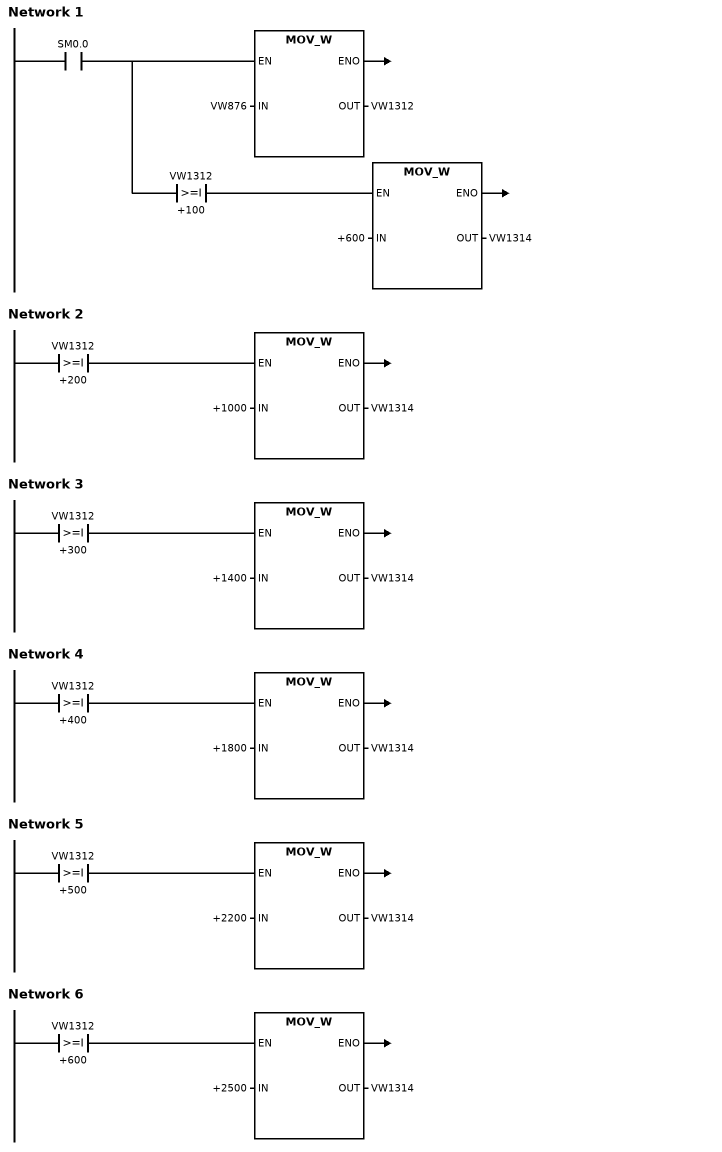
[picture p96: SBR24 networks 1-6]
Network 1
LD     SM0.0
MOVW   VW876, VW1312
AW>=   VW1312, +100
MOVW   +600, VW1314
Network 2
LDW>=  VW1312, +200
MOVW   +1000, VW1314
Network 3
LDW>=  VW1312, +300
MOVW   +1400, VW1314
Network 4
LDW>=  VW1312, +400
MOVW   +1800, VW1314
Network 5
LDW>=  VW1312, +500
MOVW   +2200, VW1314
Network 6
LDW>=  VW1312, +600
MOVW   +2500, VW1314
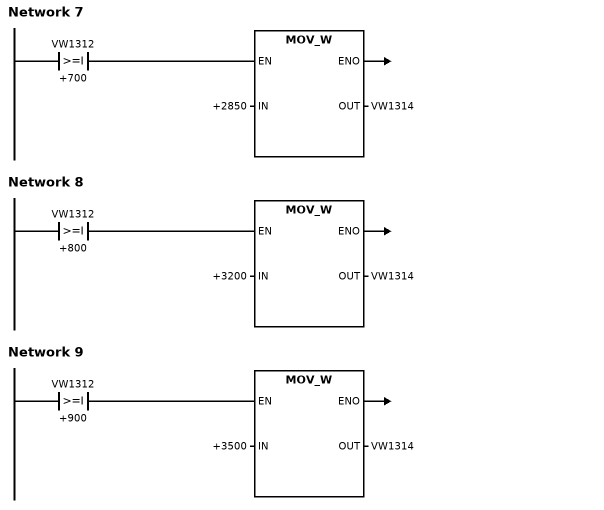
Network 7
LDW>=  VW1312, +700
MOVW   +2850, VW1314
Network 8
LDW>=  VW1312, +800
MOVW   +3200, VW1314
Network 9
LDW>=  VW1312, +900
MOVW   +3500, VW1314
END_SUBROUTINE_BLOCK

SUBROUTINE_BLOCK SprayMotorSpeedChange:SBR25
TITLE=
BEGIN
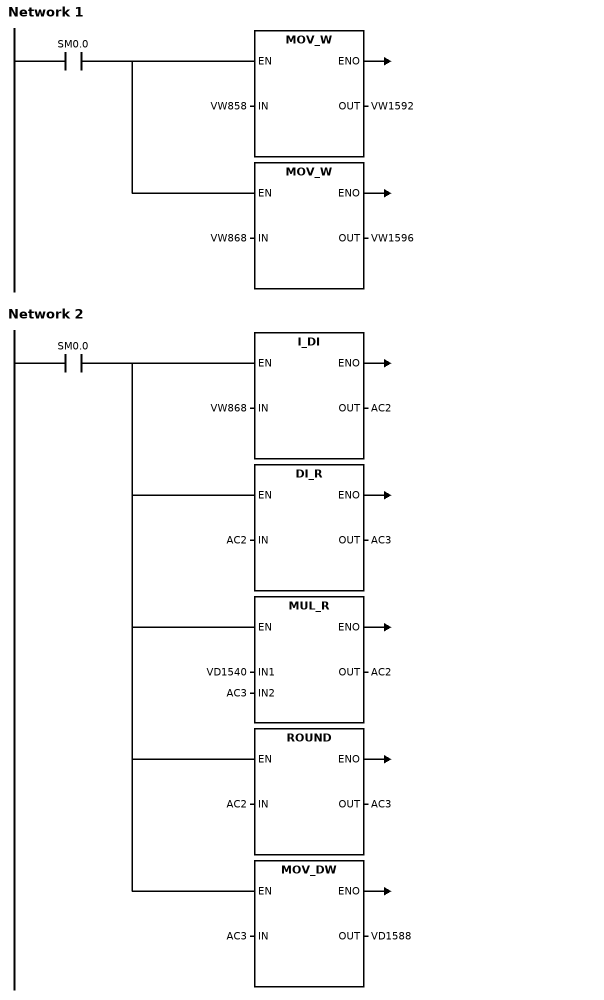
Network 1
LD     SM0.0
MOVW   VW858, VW1592
MOVW   VW868, VW1596
Network 2
LD     SM0.0
ITD    VW868, AC2
DTR    AC2, AC3
MOVR   VD1540, AC2
*R     AC3, AC2
ROUND  AC2, AC3
MOVD   AC3, VD1588
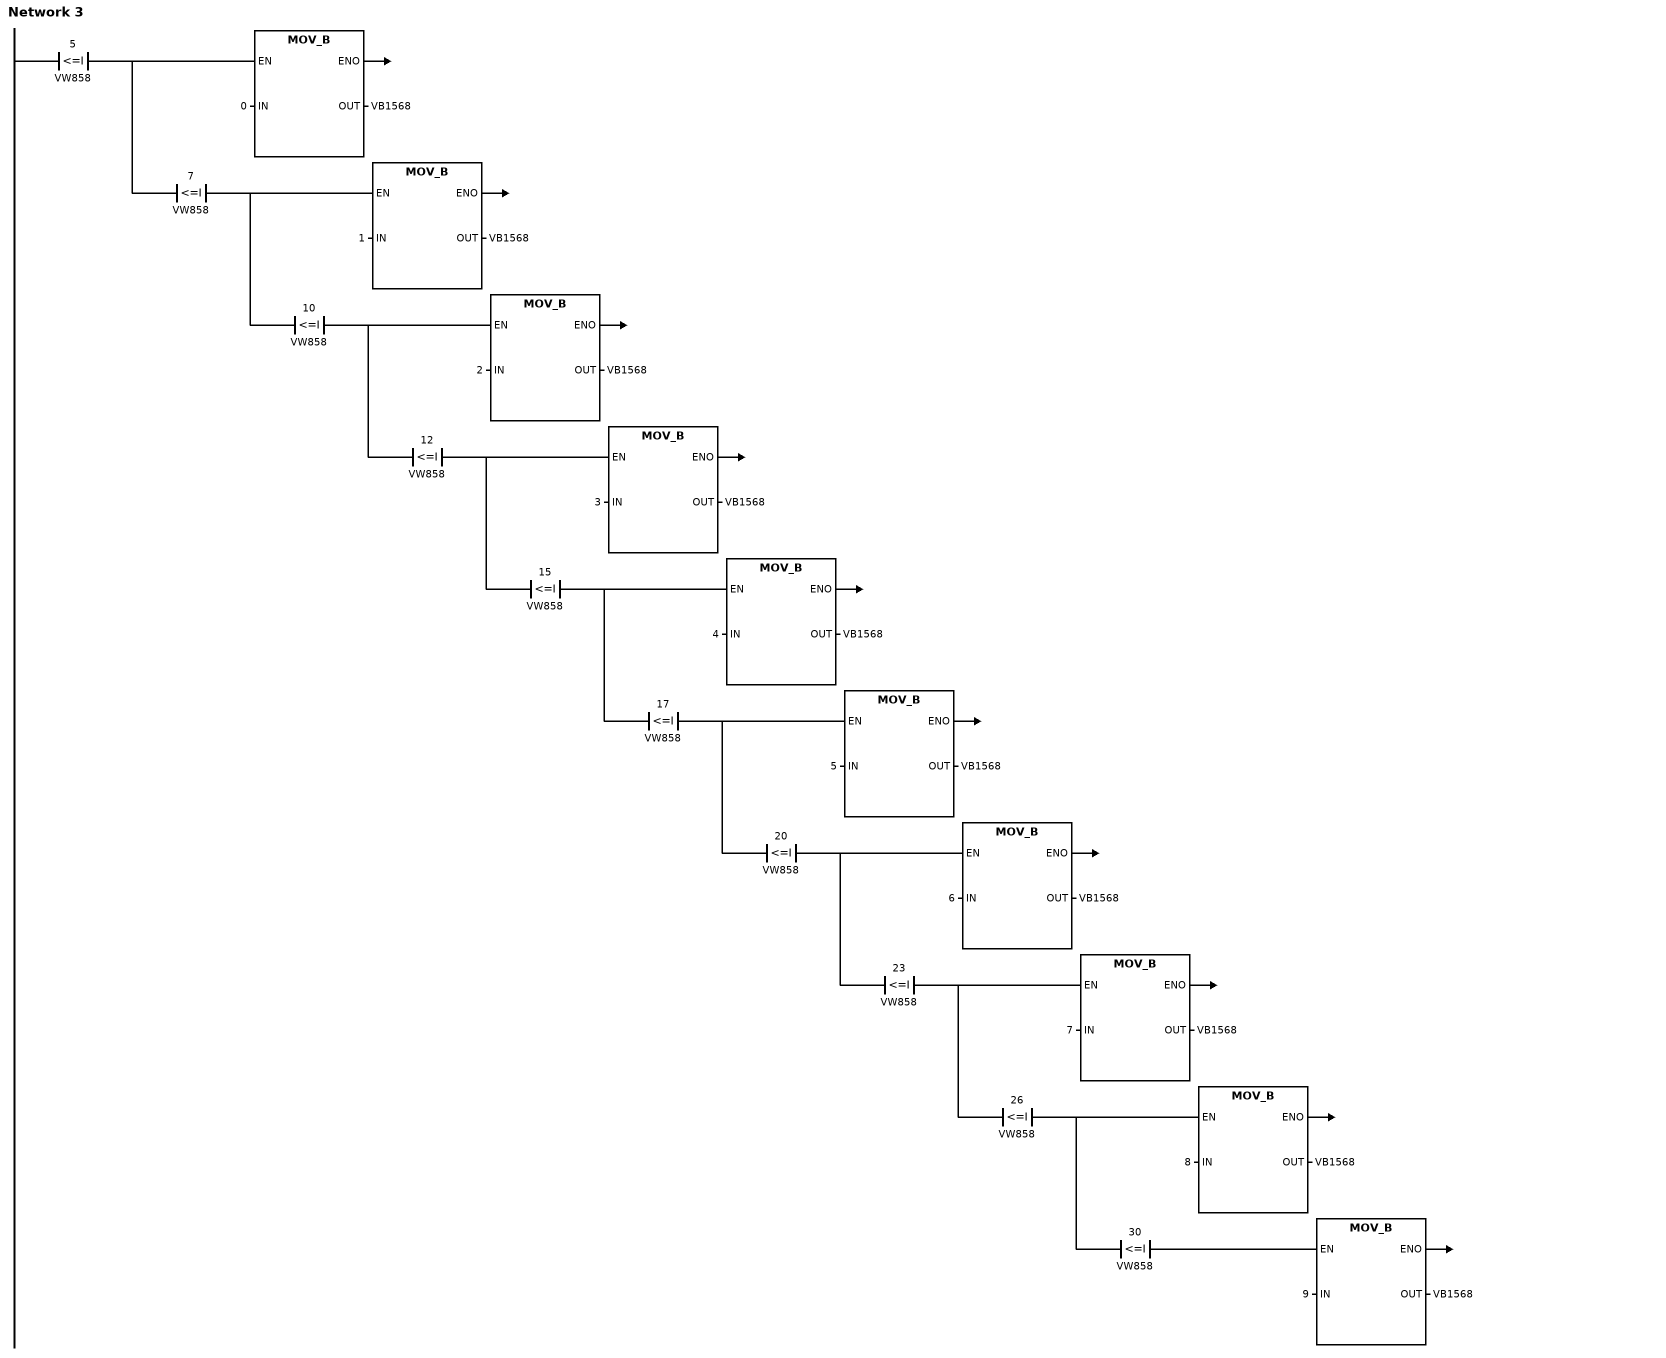
Network 3
LDW<=  5, VW858
MOVB   0, VB1568
AW<=   7, VW858
MOVB   1, VB1568
AW<=   10, VW858
MOVB   2, VB1568
AW<=   12, VW858
MOVB   3, VB1568
AW<=   15, VW858
MOVB   4, VB1568
AW<=   17, VW858
MOVB   5, VB1568
AW<=   20, VW858
MOVB   6, VB1568
AW<=   23, VW858
MOVB   7, VB1568
AW<=   26, VW858
MOVB   8, VB1568
AW<=   30, VW858
MOVB   9, VB1568
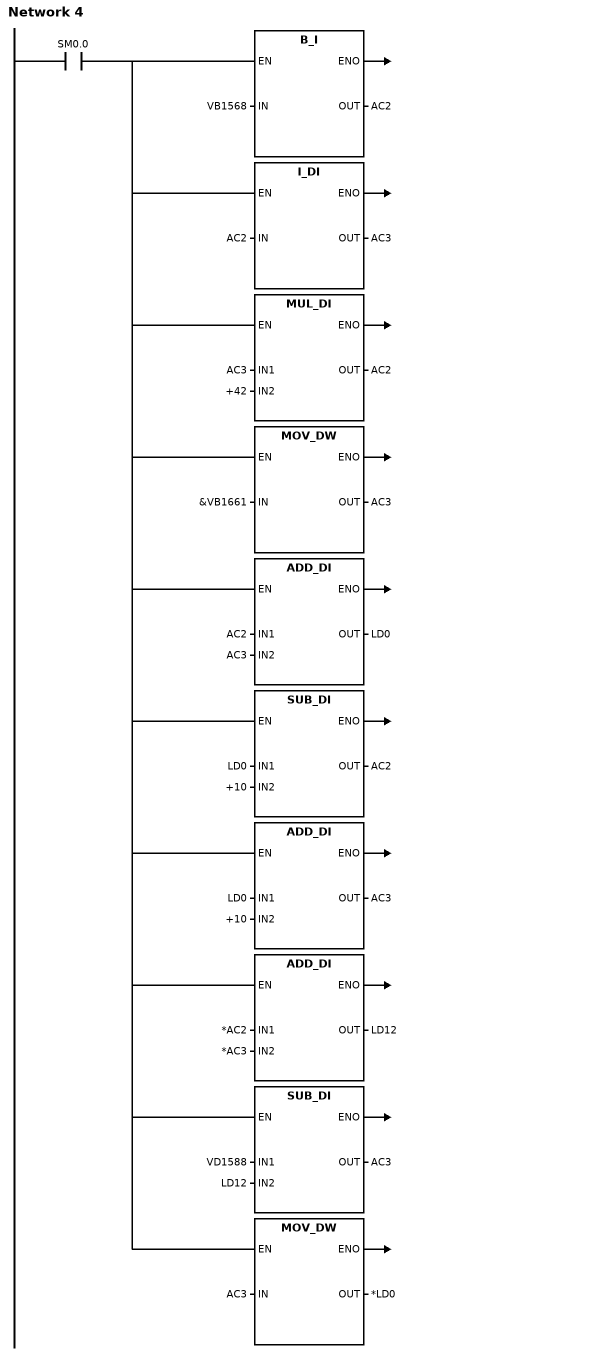
Network 4
LD     SM0.0
BTI    VB1568, AC2
ITD    AC2, AC3
MOVD   AC3, AC2
*D     +42, AC2
MOVD   &VB1661, AC3
MOVD   AC2, LD0
+D     AC3, LD0
MOVD   LD0, AC2
-D     +10, AC2
MOVD   LD0, AC3
+D     +10, AC3
MOVD   *AC2, LD12
+D     *AC3, LD12
MOVD   VD1588, AC3
-D     LD12, AC3
MOVD   AC3, *LD0
END_SUBROUTINE_BLOCK

// SBR26: protected block, not included

// SBR27: protected block, not included

// SBR28: protected block, not included

SUBROUTINE_BLOCK SysConfigure:SBR29
TITLE=SUBROUTINE COMMENTS
BEGIN
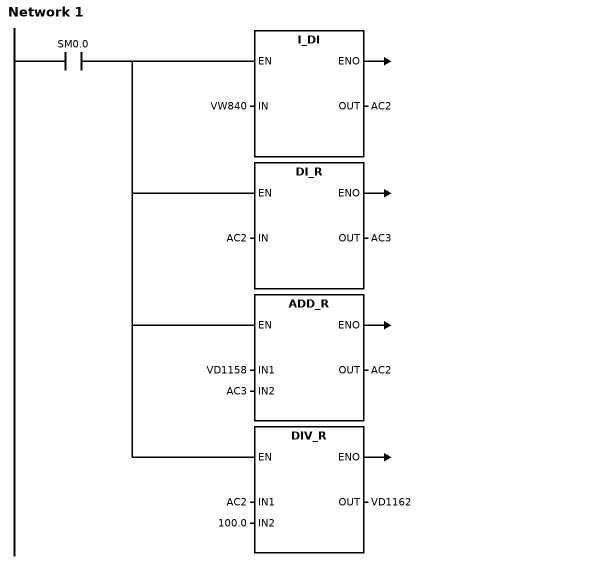
Network 1
LD     SM0.0
ITD    VW840, AC2
DTR    AC2, AC3
MOVR   VD1158, AC2
+R     AC3, AC2
MOVR   AC2, VD1162
/R     100.0, VD1162
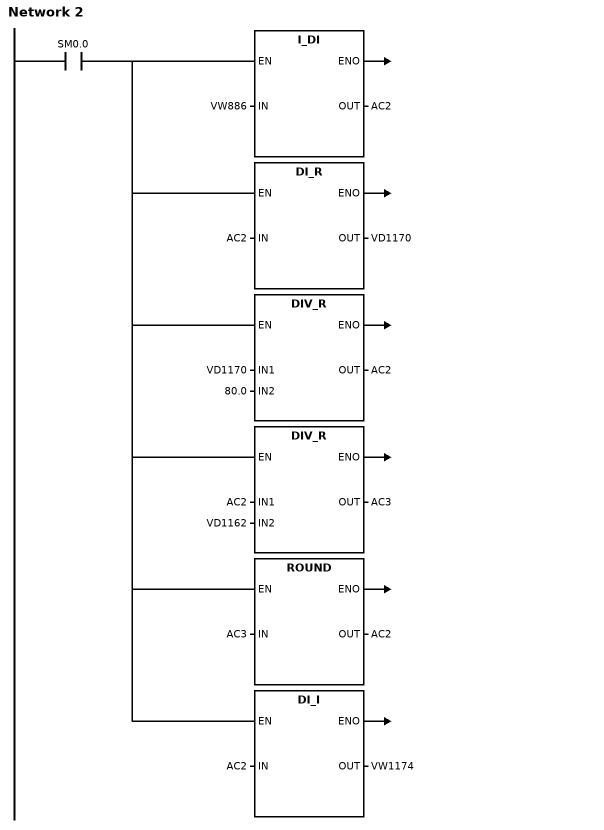
Network 2
LD     SM0.0
ITD    VW886, AC2
DTR    AC2, VD1170
MOVR   VD1170, AC2
/R     80.0, AC2
MOVR   AC2, AC3
/R     VD1162, AC3
ROUND  AC3, AC2
DTI    AC2, VW1174
END_SUBROUTINE_BLOCK

SUBROUTINE_BLOCK MyPID_M1:SBR30
TITLE=SUBROUTINE COMMENTS
VAR_INPUT
iSV:INT;	// LW0 
iPV:INT;	// LW2 
iKT:INT;	// LW4 
iKP:INT;	// LW6 
iKI:INT;	// LW8 
iKD:INT;	// LW10 
iOffset:INT;	// LW12 
pDataSave:DWORD;	// LD14 
END_VAR
VAR_OUTPUT
iPWM_1:INT;	// LW18 
chTrend:BYTE;	// LB20 
END_VAR
BEGIN
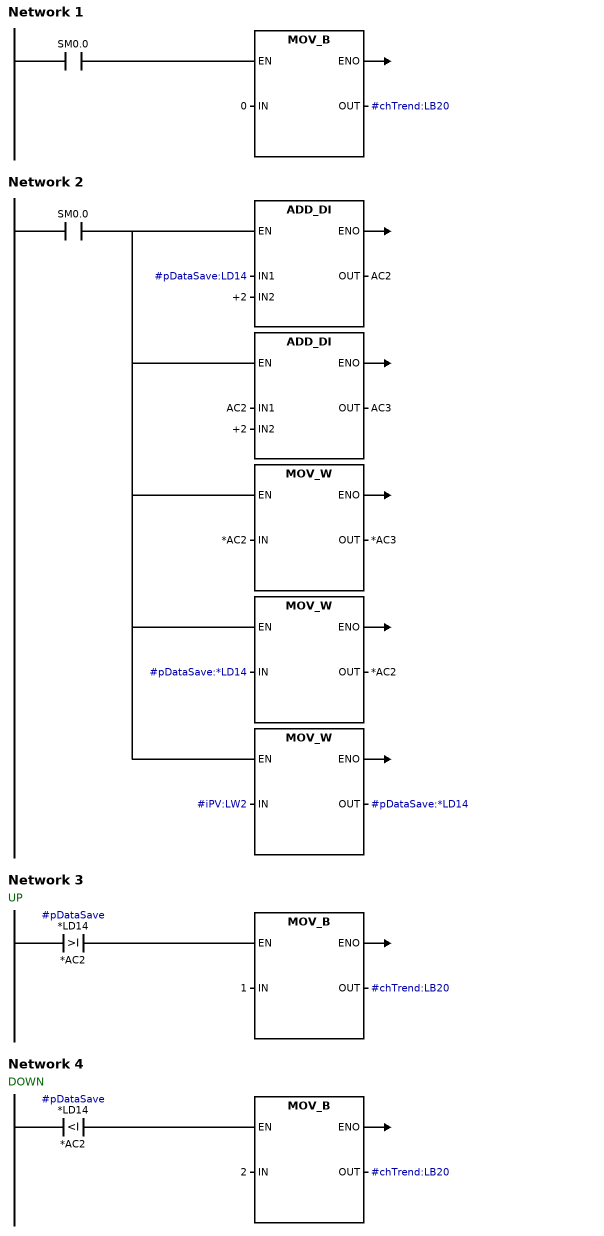
Network 1
LD     SM0.0
MOVB   0, #chTrend:LB20
Network 2
LD     SM0.0
MOVD   #pDataSave:LD14, AC2
+D     +2, AC2
MOVD   AC2, AC3
+D     +2, AC3
MOVW   *AC2, *AC3
MOVW   *#pDataSave:LD14, *AC2
MOVW   #iPV:LW2, *#pDataSave:LD14
Network 3
// UP
LDW>   *#pDataSave:LD14, *AC2
MOVB   1, #chTrend:LB20
Network 4
// DOWN
LDW<   *#pDataSave:LD14, *AC2
MOVB   2, #chTrend:LB20
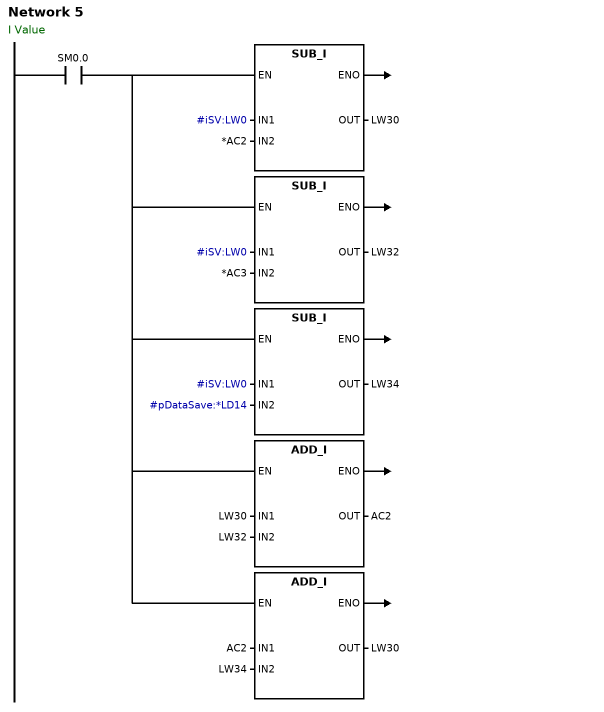
Network 5
// I Value
LD     SM0.0
MOVW   #iSV:LW0, LW30
-I     *AC2, LW30
MOVW   #iSV:LW0, LW32
-I     *AC3, LW32
MOVW   #iSV:LW0, LW34
-I     *#pDataSave:LD14, LW34
MOVW   LW30, AC2
+I     LW32, AC2
MOVW   AC2, LW30
+I     LW34, LW30
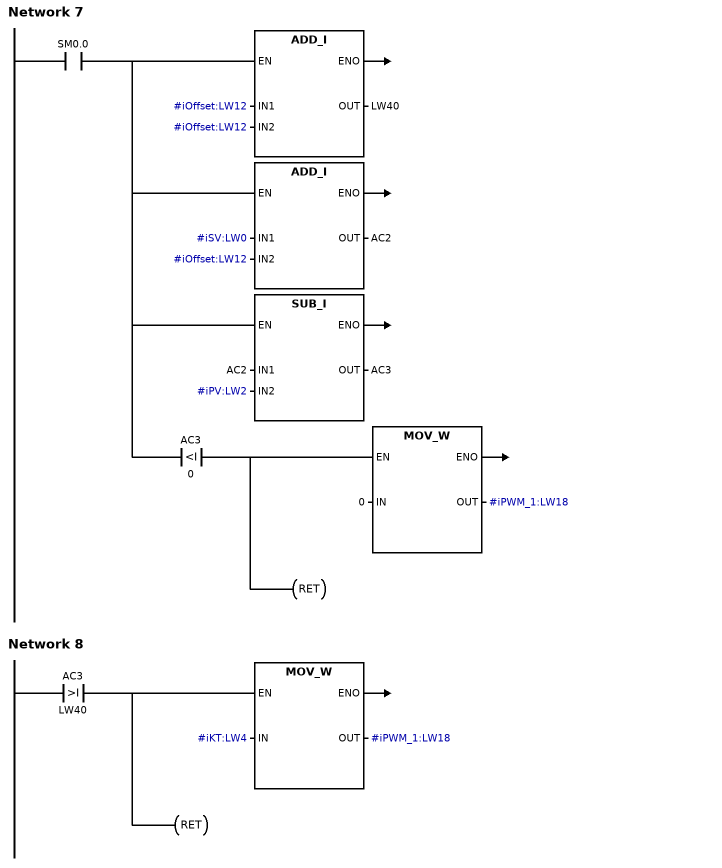
Network 7
LD     SM0.0
MOVW   #iOffset:LW12, LW40
+I     #iOffset:LW12, LW40
MOVW   #iSV:LW0, AC2
+I     #iOffset:LW12, AC2
MOVW   AC2, AC3
-I     #iPV:LW2, AC3
AW<    AC3, 0
MOVW   0, #iPWM_1:LW18
CRET
Network 8
LDW>   AC3, LW40
MOVW   #iKT:LW4, #iPWM_1:LW18
CRET
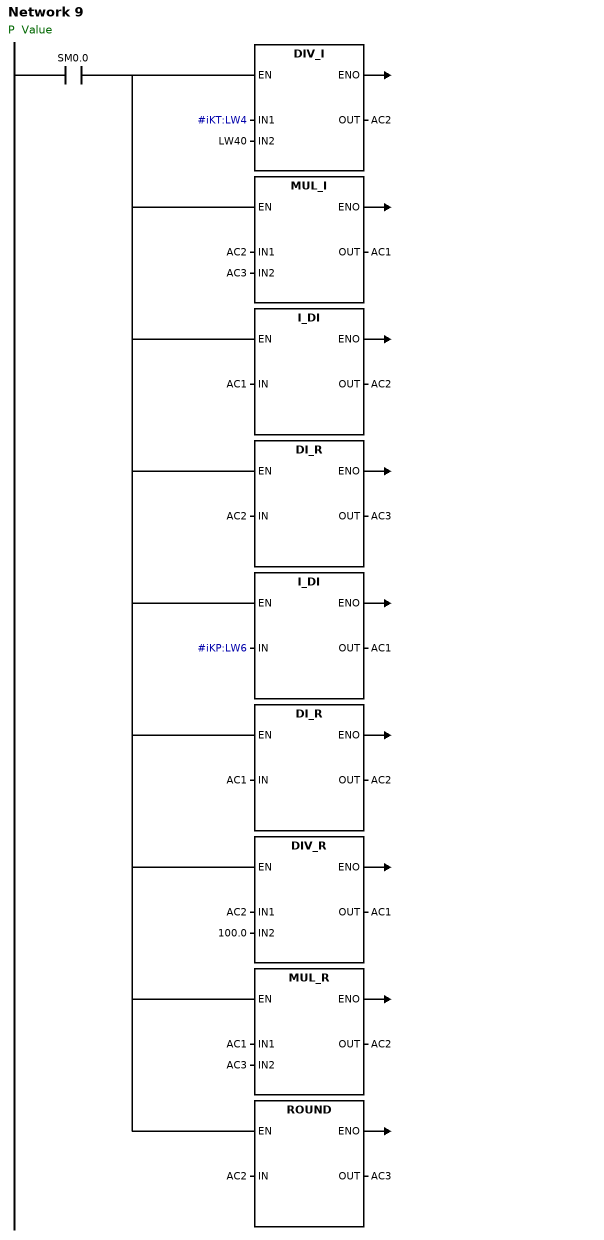
Network 9
// P  Value
LD     SM0.0
MOVW   #iKT:LW4, AC2
/I     LW40, AC2
MOVW   AC2, AC1
*I     AC3, AC1
ITD    AC1, AC2
DTR    AC2, AC3
ITD    #iKP:LW6, AC1
DTR    AC1, AC2
MOVR   AC2, AC1
/R     100.0, AC1
MOVR   AC1, AC2
*R     AC3, AC2
ROUND  AC2, AC3
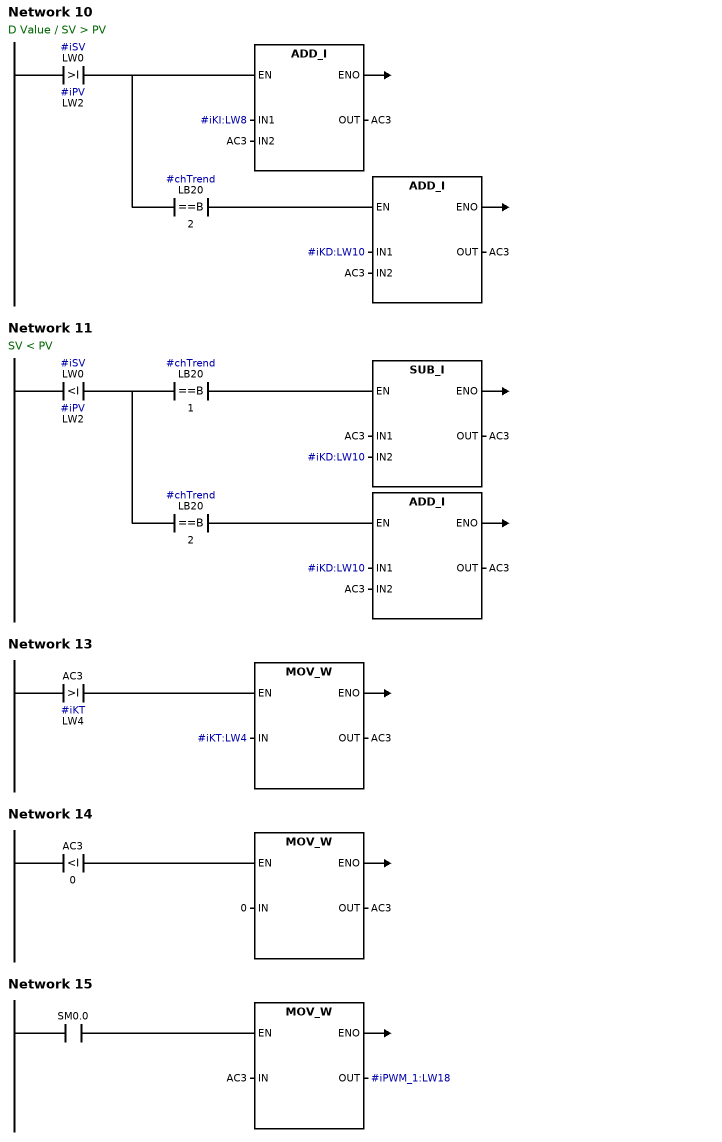
Network 10
// D Value
// SV > PV
LDW>   #iSV:LW0, #iPV:LW2
+I     #iKI:LW8, AC3
AB=    #chTrend:LB20, 2
+I     #iKD:LW10, AC3
Network 11
// SV < PV
LDW<   #iSV:LW0, #iPV:LW2
LPS
AB=    #chTrend:LB20, 1
-I     #iKD:LW10, AC3
LPP
AB=    #chTrend:LB20, 2
+I     #iKD:LW10, AC3
Network 12
// I????
Network 13
LDW>   AC3, #iKT:LW4
MOVW   #iKT:LW4, AC3
Network 14
LDW<   AC3, 0
MOVW   0, AC3
Network 15
LD     SM0.0
MOVW   AC3, #iPWM_1:LW18
END_SUBROUTINE_BLOCK

SUBROUTINE_BLOCK StopQ1Pulse:SBR31
TITLE=SUBROUTINE COMMENTS
BEGIN
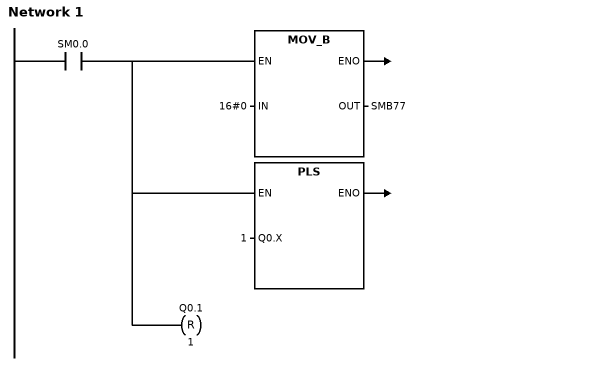
Network 1
LD     SM0.0
MOVB   16#0, SMB77
PLS    1
R      Q0.1, 1
END_SUBROUTINE_BLOCK

SUBROUTINE_BLOCK WidthPulseVB4000_4099:SBR32
TITLE=SUBROUTINE COMMENTS
VAR_INPUT
iPCBWidth:INT;	// LW0 
iSpeedHz:INT;	// LW2 
END_VAR
BEGIN
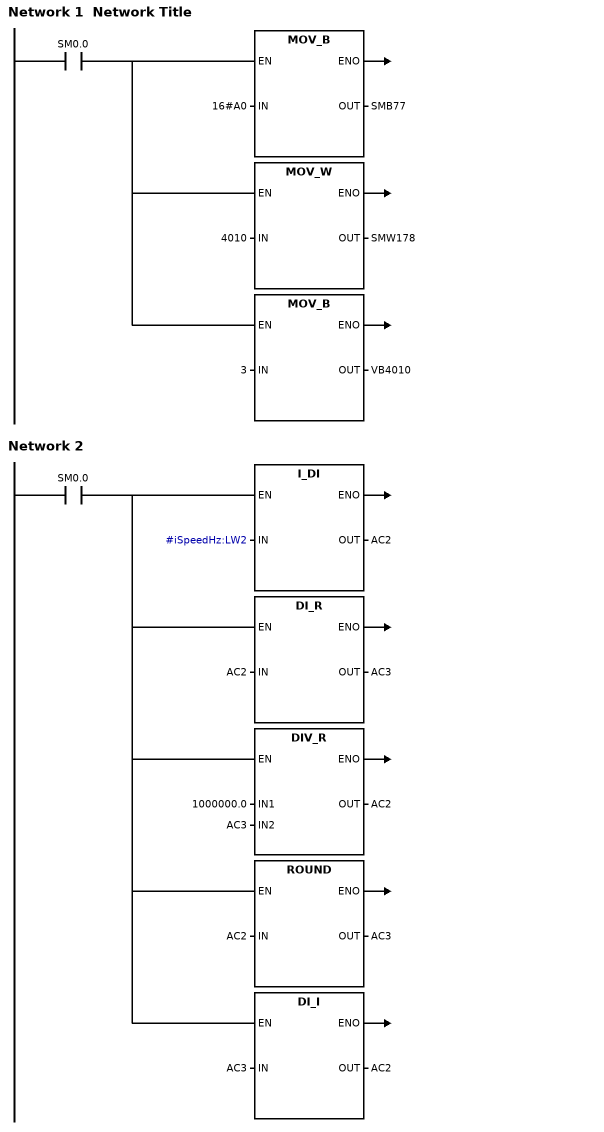
Network 1 // Network Title
LD     SM0.0
MOVB   16#A0, SMB77
MOVW   4010, SMW178
MOVB   3, VB4010
Network 2
LD     SM0.0
ITD    #iSpeedHz:LW2, AC2
DTR    AC2, AC3
MOVR   1000000.0, AC2
/R     AC3, AC2
ROUND  AC2, AC3
DTI    AC3, AC2
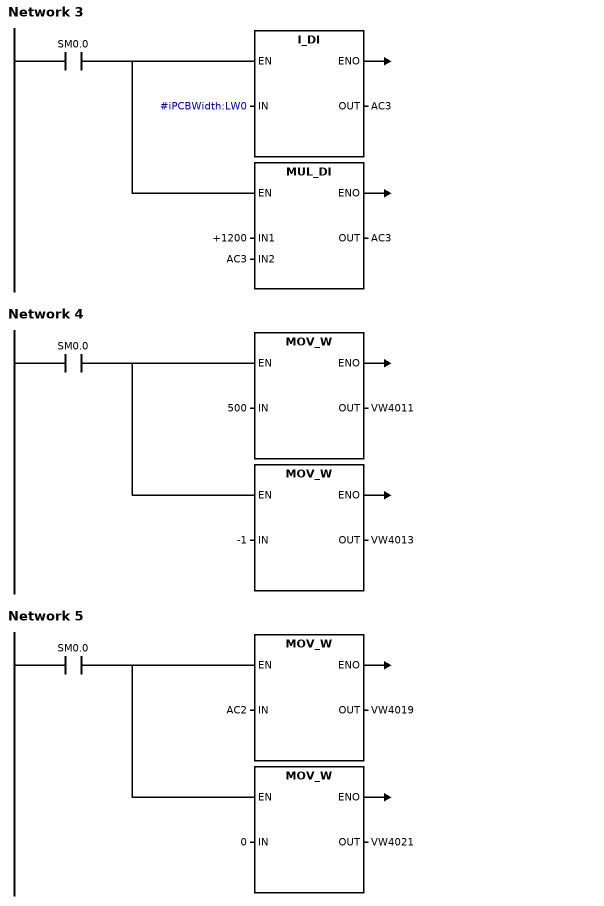
Network 3
LD     SM0.0
ITD    #iPCBWidth:LW0, AC3
*D     +1200, AC3
Network 4
LD     SM0.0
MOVW   500, VW4011
MOVW   -1, VW4013
Network 5
LD     SM0.0
MOVW   AC2, VW4019
MOVW   0, VW4021
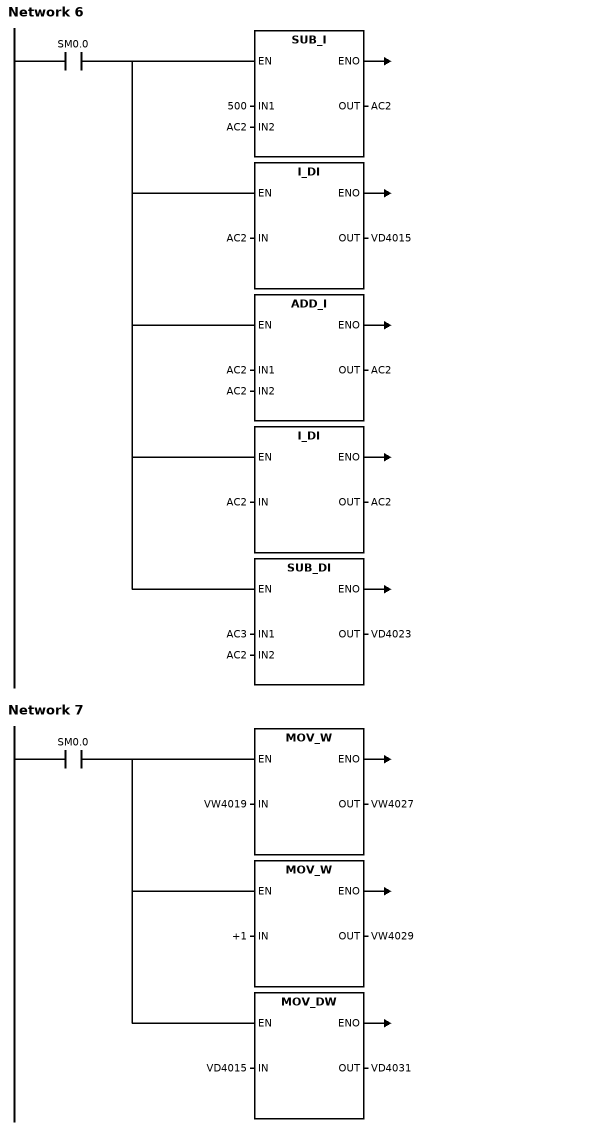
Network 6
LD     SM0.0
INVW   AC2
INCW   AC2
+I     500, AC2
ITD    AC2, VD4015
+I     AC2, AC2
ITD    AC2, AC2
MOVD   AC3, VD4023
-D     AC2, VD4023
Network 7
LD     SM0.0
MOVW   VW4019, VW4027
MOVW   +1, VW4029
MOVD   VD4015, VD4031
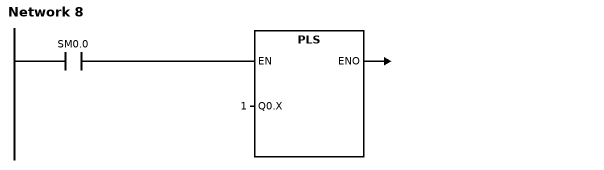
Network 8
LD     SM0.0
PLS    1
END_SUBROUTINE_BLOCK

SUBROUTINE_BLOCK TimerFlagVB600_699:SBR33
TITLE=SUBROUTINE COMMENTS
BEGIN
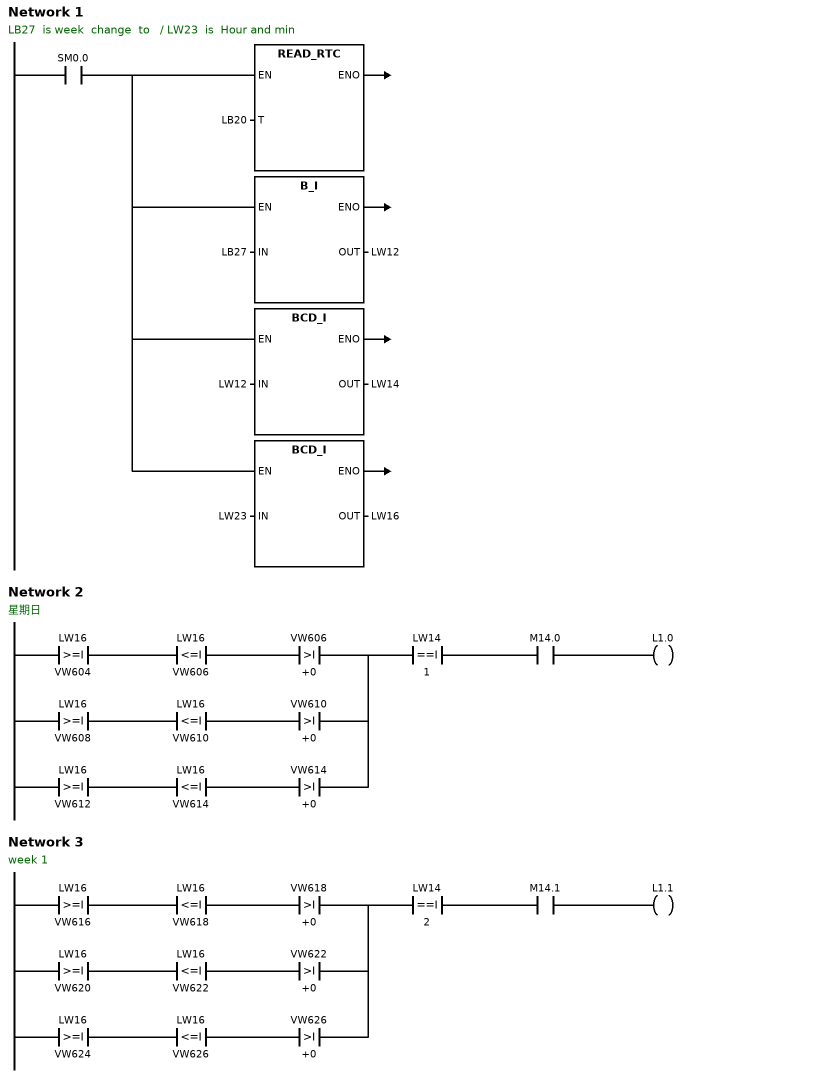
Network 1
// LB27  is week  change  to  
// LW23  is  Hour and min
LD     SM0.0
TODR   LB20
BTI    LB27, LW12
MOVW   LW12, LW14
BCDI   LW14
MOVW   LW23, LW16
BCDI   LW16
Network 2
// 星期日
LDW>=  LW16, VW604
AW<=   LW16, VW606
AW>    VW606, +0
LDW>=  LW16, VW608
AW<=   LW16, VW610
AW>    VW610, +0
OLD
LDW>=  LW16, VW612
AW<=   LW16, VW614
AW>    VW614, +0
OLD
AW=    LW14, 1
A      M14.0
=      L1.0
Network 3
// week 1
LDW>=  LW16, VW616
AW<=   LW16, VW618
AW>    VW618, +0
LDW>=  LW16, VW620
AW<=   LW16, VW622
AW>    VW622, +0
OLD
LDW>=  LW16, VW624
AW<=   LW16, VW626
AW>    VW626, +0
OLD
AW=    LW14, 2
A      M14.1
=      L1.1
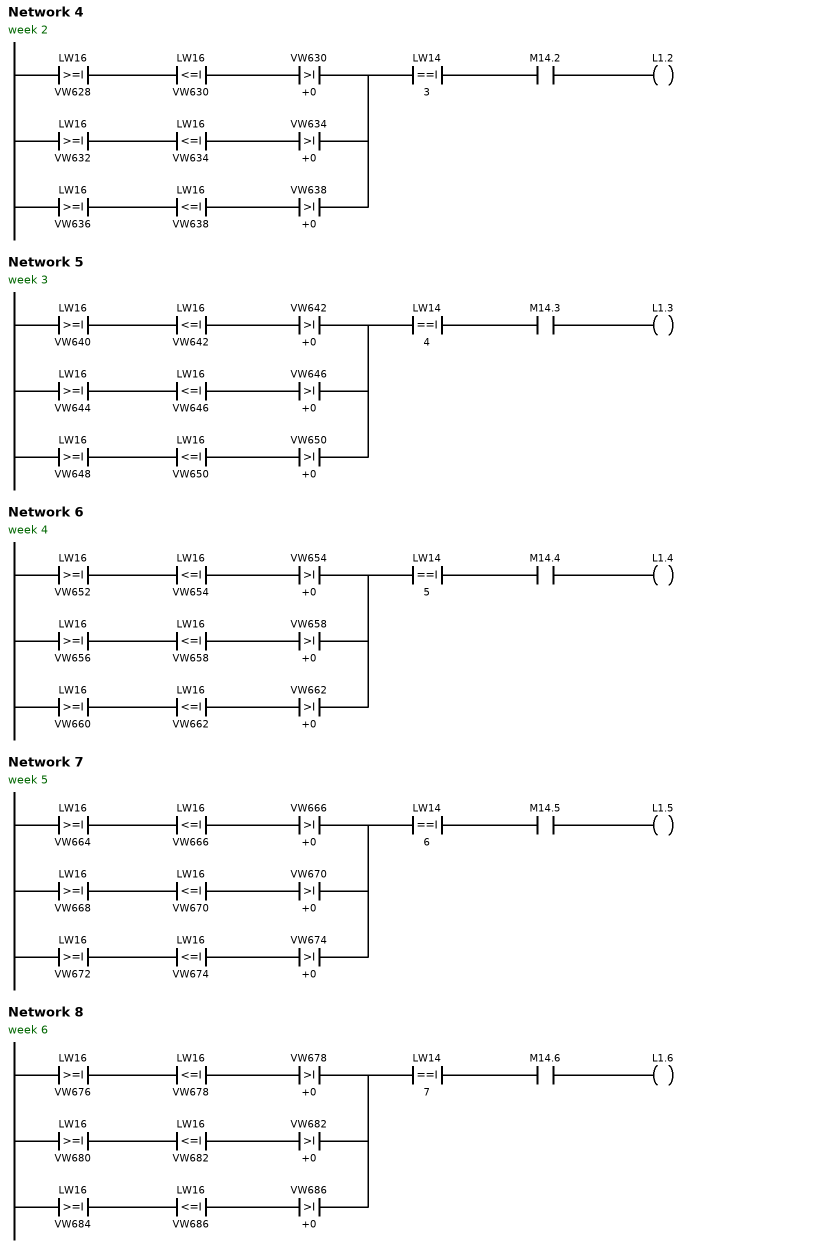
Network 4
// week 2
LDW>=  LW16, VW628
AW<=   LW16, VW630
AW>    VW630, +0
LDW>=  LW16, VW632
AW<=   LW16, VW634
AW>    VW634, +0
OLD
LDW>=  LW16, VW636
AW<=   LW16, VW638
AW>    VW638, +0
OLD
AW=    LW14, 3
A      M14.2
=      L1.2
Network 5
// week 3
LDW>=  LW16, VW640
AW<=   LW16, VW642
AW>    VW642, +0
LDW>=  LW16, VW644
AW<=   LW16, VW646
AW>    VW646, +0
OLD
LDW>=  LW16, VW648
AW<=   LW16, VW650
AW>    VW650, +0
OLD
AW=    LW14, 4
A      M14.3
=      L1.3
Network 6
// week 4
LDW>=  LW16, VW652
AW<=   LW16, VW654
AW>    VW654, +0
LDW>=  LW16, VW656
AW<=   LW16, VW658
AW>    VW658, +0
OLD
LDW>=  LW16, VW660
AW<=   LW16, VW662
AW>    VW662, +0
OLD
AW=    LW14, 5
A      M14.4
=      L1.4
Network 7
// week 5
LDW>=  LW16, VW664
AW<=   LW16, VW666
AW>    VW666, +0
LDW>=  LW16, VW668
AW<=   LW16, VW670
AW>    VW670, +0
OLD
LDW>=  LW16, VW672
AW<=   LW16, VW674
AW>    VW674, +0
OLD
AW=    LW14, 6
A      M14.5
=      L1.5
Network 8
// week 6
LDW>=  LW16, VW676
AW<=   LW16, VW678
AW>    VW678, +0
LDW>=  LW16, VW680
AW<=   LW16, VW682
AW>    VW682, +0
OLD
LDW>=  LW16, VW684
AW<=   LW16, VW686
AW>    VW686, +0
OLD
AW=    LW14, 7
A      M14.6
=      L1.6
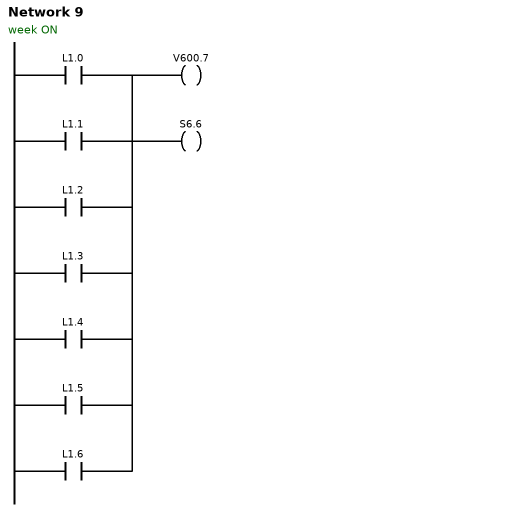
Network 9
// week ON
LD     L1.0
O      L1.1
O      L1.2
O      L1.3
O      L1.4
O      L1.5
O      L1.6
=      V600.7
=      S6.6
END_SUBROUTINE_BLOCK

SUBROUTINE_BLOCK Preheart_equalize:SBR34
TITLE=WaveSpewWagVB1300_1319//T160_T164
BEGIN
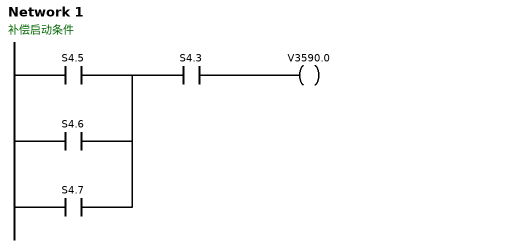
Network 1
// 补偿启动条件
LD     S4.5
O      S4.6
O      S4.7
A      S4.3
=      V3590.0
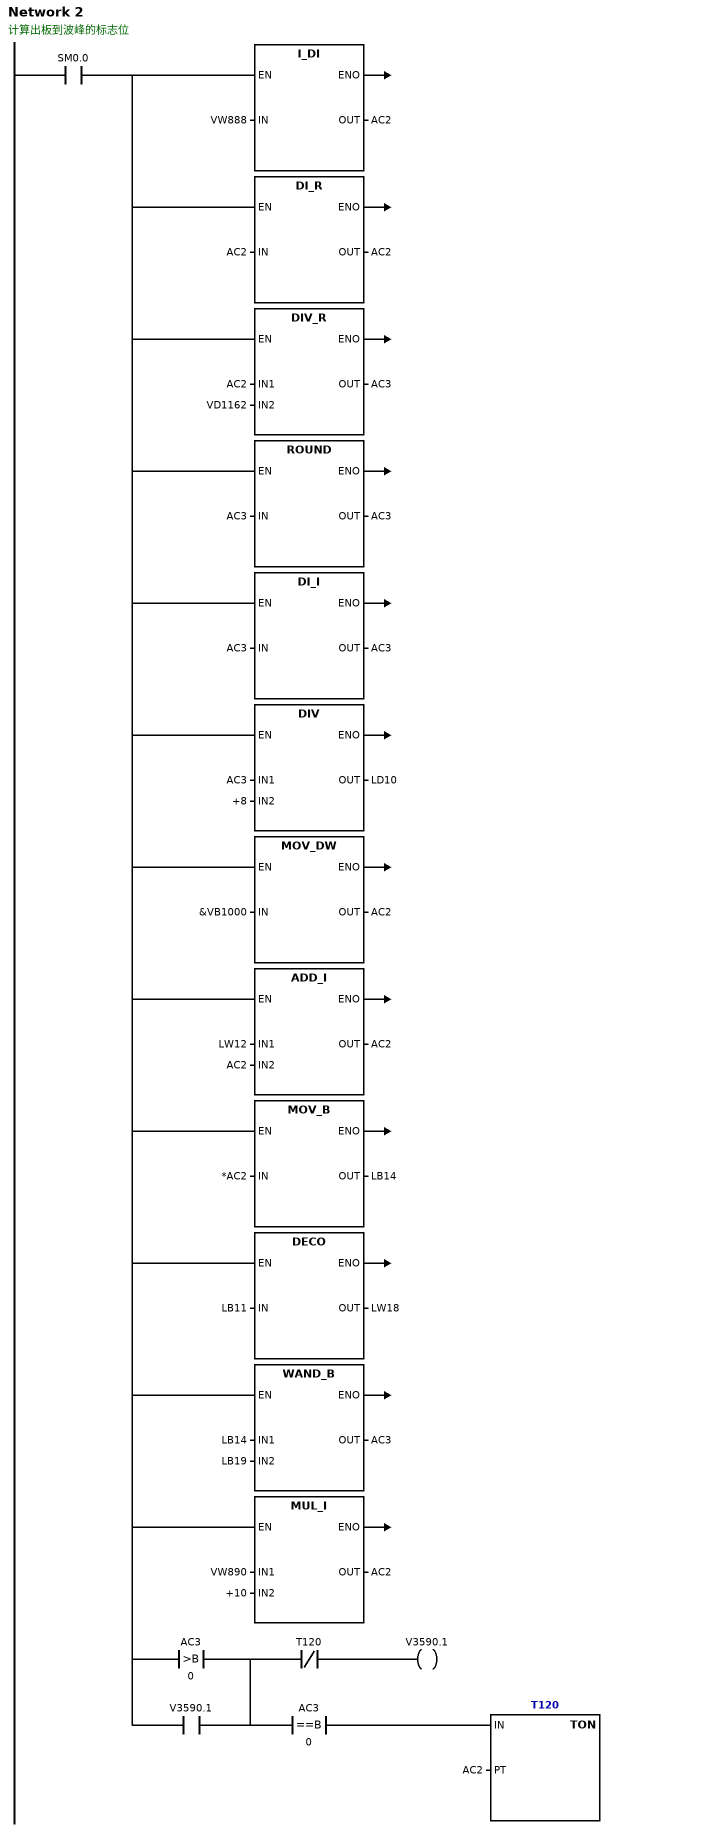
Network 2
// 计算出板到波峰的标志位
LD     SM0.0
ITD    VW888, AC2
DTR    AC2, AC2
MOVR   AC2, AC3
/R     VD1162, AC3
ROUND  AC3, AC3
DTI    AC3, AC3
MOVW   AC3, LW12
DIV    +8, LD10
MOVD   &VB1000, AC2
+I     LW12, AC2
MOVB   *AC2, LB14
DECO   LB11, LW18
MOVB   LB14, AC3
ANDB   LB19, AC3
MOVW   VW890, AC2
*I     +10, AC2
LDB>   AC3, 0
O      V3590.1
ALD
LPS
AN     T120
=      V3590.1
LPP
AB=    AC3, 0
TON    T120, AC2
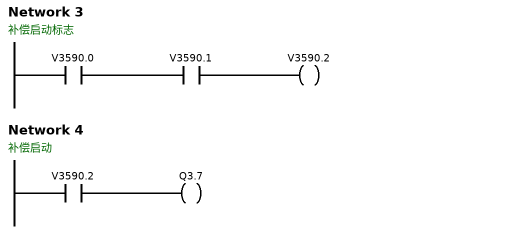
Network 3
// 补偿启动标志
LD     V3590.0
A      V3590.1
=      V3590.2
Network 4
// 补偿启动
LD     V3590.2
=      Q3.7
Network 5 // 网络标题
// 网络注释
Network 15 // 网络标题
// 网络注释
Network 25 // Network Title
// Network Comment
END_SUBROUTINE_BLOCK

SUBROUTINE_BLOCK PCB_Block:SBR45
TITLE=子程序注释
BEGIN
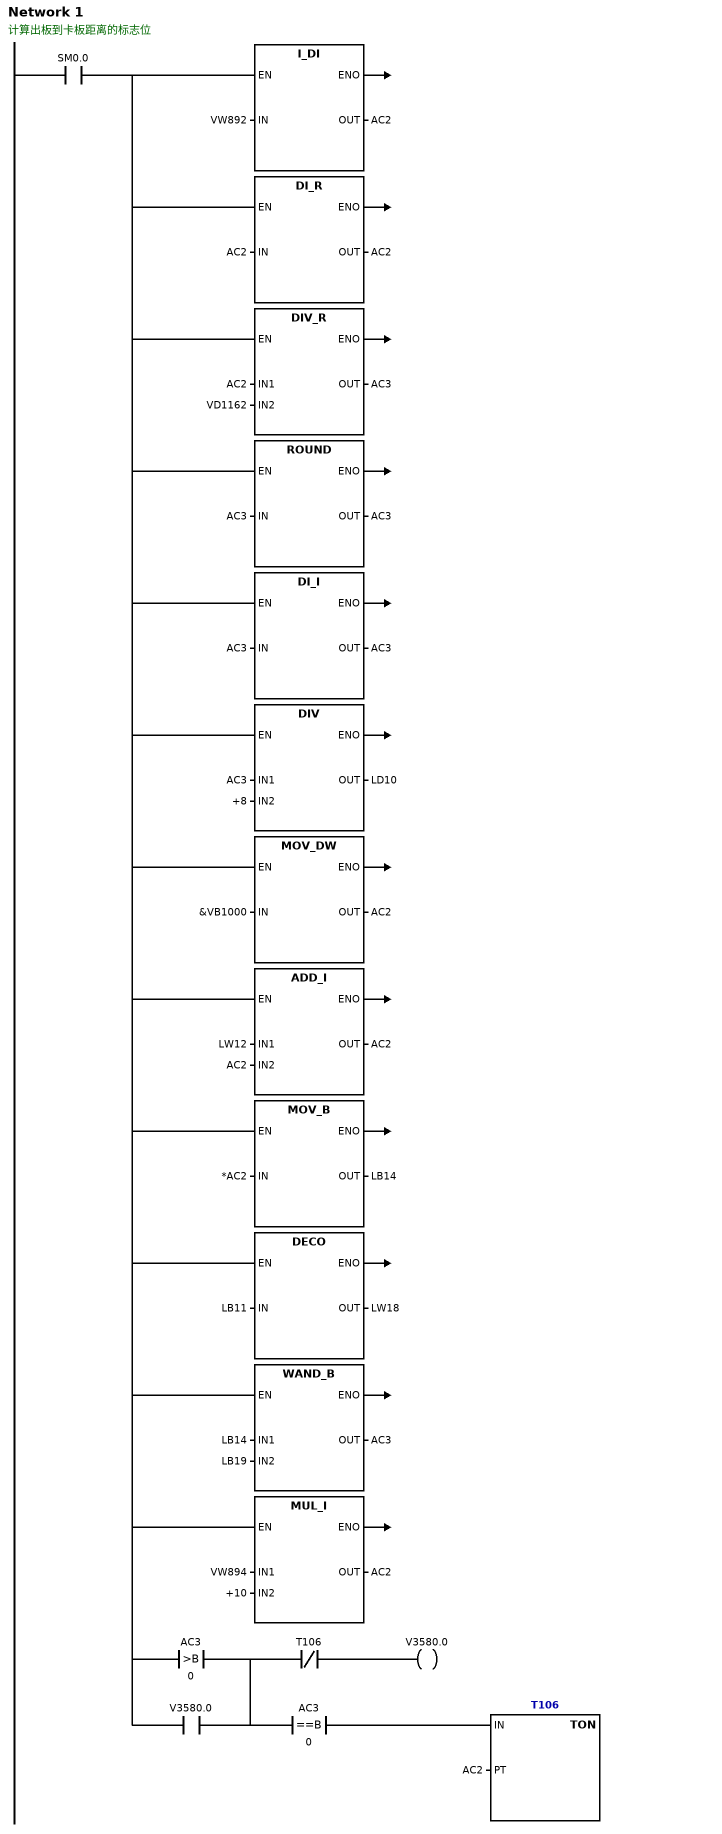
Network 1
// 计算出板到卡板距离的标志位
LD     SM0.0
ITD    VW892, AC2
DTR    AC2, AC2
MOVR   AC2, AC3
/R     VD1162, AC3
ROUND  AC3, AC3
DTI    AC3, AC3
MOVW   AC3, LW12
DIV    +8, LD10
MOVD   &VB1000, AC2
+I     LW12, AC2
MOVB   *AC2, LB14
DECO   LB11, LW18
MOVB   LB14, AC3
ANDB   LB19, AC3
MOVW   VW894, AC2
*I     +10, AC2
LDB>   AC3, 0
O      V3580.0
ALD
LPS
AN     T106
=      V3580.0
LPP
AB=    AC3, 0
TON    T106, AC2
